{attribute 'GeneratedUsingTerminal: EP9128-0021-0017'}
{attribute addProperty BoxType "EP9128-0021-0017"}
{attribute addProperty Id "A_0010_EP9128_0021_0018A_0010_EP9128_0021_0018_C959F4E2583A_0007_EP9128_0021_0017_2_EP9128_1021EP9128_1FC0878B2A_0007_EP9128_0021_0017_3_EP9128_2021EP9128_1FC0878B2"}
{attribute addProperty CRC "4182334792"}
{attribute addProperty Size "587"}
TYPE A_0007_EP9128_0021_0017_F9495D48 EXTENDS EP9128_1FC0878B :
STRUCT
	{attribute addProperty Name "A_0010(EP9128-0021-0018)"}
	{attribute addProperty PreviousPort "A_0007(EP9128-0021-0017) : D"}
	A_0010_EP9128_0021_0018 : A_0010_EP9128_0021_0018_C959F4E2;
	{attribute addProperty Name "A_0007(EP9128-0021-0017)_2 (EP9128-1021)"}
	{attribute addProperty PreviousPort "A_0007(EP9128-0021-0017) : C"}
	A_0007_EP9128_0021_0017_2_EP9128_1021 : EP9128_1FC0878B;
	{attribute addProperty Name "A_0007(EP9128-0021-0017)_3 (EP9128-2021)"}
	{attribute addProperty PreviousPort "A_0007(EP9128-0021-0017)_2 (EP9128-1021) : C"}
	A_0007_EP9128_0021_0017_3_EP9128_2021 : EP9128_1FC0878B;
END_STRUCT
END_TYPE

(* stored: Version 1.2.0.0, ProductVersion 3.1.4024.9
   DUT A_0007_EP9128_0021_0017_F9495D48: Id {993079e5-2326-45b3-b2b5-1523a47c00d4} *)
